{attribute 'GeneratedUsingTerminal: IODEVICETYPE_ETHERCATPROT'}
{attribute addProperty BoxType "IODEVICETYPE_ETHERCATPROT"}
{attribute addProperty Id "Beckhoff_EL1xxxBeckhoff_EL1xxx_3E37AACA6236Beckhoff_EL2xxxBeckhoff_EL2xxx_F4C539CA2992Beckhoff_EL3xxxBeckhoff_EL3xxx_05984D3D1813Beckhoff_EL3xxx_0030Beckhoff_EL3xxx_0030_C37B7D48265Beckhoff_EL4xxxBeckhoff_EL4xxx_44DCAF8D2405Beckhoff_EL5xxxBeckhoff_EL5xxx_A510F2723086Beckhoff_EL6xxxBeckhoff_EL6xxx_5832F4A84115Beckhoff_EL7xxxBeckhoff_EL7xxx_96878FD52666Beckhoff_EL9xxxBeckhoff_EL9xxx_6E572B5F1254Beckhoff_EL15xxBeckhoff_EL15xx_7FFDF3B3529Beckhoff_EL19xxBeckhoff_EL19xx_C9550BF750Beckhoff_EL25xxBeckhoff_EL25xx_A1E3F9182720Beckhoff_EL29xxBeckhoff_EL29xx_FCC67B4476Beckhoff_EL30xxBeckhoff_EL30xx_59D865295129Beckhoff_EL31xxBeckhoff_EL31xx_098DC56E3694Beckhoff_EL32xxBeckhoff_EL32xx_A91E9D412581Beckhoff_EL33xxBeckhoff_EL33xx_149C8FF52459Beckhoff_EL34xxBeckhoff_EL34xx_5C8507D711825Beckhoff_EL37xxBeckhoff_EL37xx_82AB11DA2253Beckhoff_EL47xxBeckhoff_EL47xx_F9F61196294Beckhoff_EL66xxBeckhoff_EL66xx_32F43B791034Beckhoff_EL67xxBeckhoff_EL67xx_9D033AAA966Beckhoff_EL68xxBeckhoff_EL68xx_6F2062753597Beckhoff_EL69xxBeckhoff_EL69xx_55DE5C9C198Beckhoff_EL72xxBeckhoff_EL72xx_566ED46D3383Beckhoff_EL73xxBeckhoff_EL73xx_3D4E24E01278Beckhoff_EL99xxBeckhoff_EL99xx_FA66A12D10SyncUnitsSyncUnits_9F8710E11242InputsInputs_25A0042B160OutputsOutputs_2397A10E106InfoDataInfoData_E68C61CD28"}
{attribute addProperty CRC "3501869254"}
{attribute addProperty Size "68444"}
TYPE EtherCAT_Master_ELxxxx_D0BA48C6 EXTENDS EtcMasterBase_62654B43 :
STRUCT
	{attribute addProperty Name "Beckhoff EL1xxx"}
	{attribute addProperty PreviousPort "EtherCAT_Master_ELxxxx : Master"}
	Beckhoff_EL1xxx : Beckhoff_EL1xxx_3E37AACA;
	{attribute addProperty Name "Beckhoff EL2xxx"}
	{attribute addProperty PreviousPort "Beckhoff EL1xxx : C"}
	Beckhoff_EL2xxx : Beckhoff_EL2xxx_F4C539CA;
	{attribute addProperty Name "Beckhoff EL3xxx"}
	{attribute addProperty PreviousPort "Beckhoff EL2xxx : C"}
	Beckhoff_EL3xxx : Beckhoff_EL3xxx_05984D3D;
	{attribute addProperty Name "Beckhoff EL3xxx-0030"}
	{attribute addProperty PreviousPort "Beckhoff EL3xxx : C"}
	Beckhoff_EL3xxx_0030 : Beckhoff_EL3xxx_0030_C37B7D48;
	{attribute addProperty Name "Beckhoff EL4xxx"}
	{attribute addProperty PreviousPort "Beckhoff EL3xxx-0030 : C"}
	Beckhoff_EL4xxx : Beckhoff_EL4xxx_44DCAF8D;
	{attribute addProperty Name "Beckhoff EL5xxx"}
	{attribute addProperty PreviousPort "Beckhoff EL4xxx : C"}
	Beckhoff_EL5xxx : Beckhoff_EL5xxx_A510F272;
	{attribute addProperty Name "Beckhoff EL6xxx"}
	{attribute addProperty PreviousPort "Beckhoff EL5xxx : C"}
	Beckhoff_EL6xxx : Beckhoff_EL6xxx_5832F4A8;
	{attribute addProperty Name "Beckhoff EL7xxx"}
	{attribute addProperty PreviousPort "Beckhoff EL6xxx : C"}
	Beckhoff_EL7xxx : Beckhoff_EL7xxx_96878FD5;
	{attribute addProperty Name "Beckhoff EL9xxx"}
	{attribute addProperty PreviousPort "Beckhoff EL7xxx : C"}
	Beckhoff_EL9xxx : Beckhoff_EL9xxx_6E572B5F;
	{attribute addProperty Name "Beckhoff EL15xx"}
	{attribute addProperty PreviousPort "Beckhoff EL9xxx : C"}
	Beckhoff_EL15xx : Beckhoff_EL15xx_7FFDF3B3;
	{attribute addProperty Name "Beckhoff EL19xx"}
	{attribute addProperty PreviousPort "Beckhoff EL15xx : C"}
	Beckhoff_EL19xx : Beckhoff_EL19xx_C9550BF7;
	{attribute addProperty Name "Beckhoff EL25xx"}
	{attribute addProperty PreviousPort "Beckhoff EL19xx : C"}
	Beckhoff_EL25xx : Beckhoff_EL25xx_A1E3F918;
	{attribute addProperty Name "Beckhoff EL29xx"}
	{attribute addProperty PreviousPort "Beckhoff EL25xx : C"}
	Beckhoff_EL29xx : Beckhoff_EL29xx_FCC67B44;
	{attribute addProperty Name "Beckhoff EL30xx"}
	{attribute addProperty PreviousPort "Beckhoff EL29xx : C"}
	Beckhoff_EL30xx : Beckhoff_EL30xx_59D86529;
	{attribute addProperty Name "Beckhoff EL31xx"}
	{attribute addProperty PreviousPort "Beckhoff EL30xx : C"}
	Beckhoff_EL31xx : Beckhoff_EL31xx_098DC56E;
	{attribute addProperty Name "Beckhoff EL32xx"}
	{attribute addProperty PreviousPort "Beckhoff EL31xx : C"}
	Beckhoff_EL32xx : Beckhoff_EL32xx_A91E9D41;
	{attribute addProperty Name "Beckhoff EL33xx"}
	{attribute addProperty PreviousPort "Beckhoff EL32xx : C"}
	Beckhoff_EL33xx : Beckhoff_EL33xx_149C8FF5;
	{attribute addProperty Name "Beckhoff EL34xx"}
	{attribute addProperty PreviousPort "Beckhoff EL33xx : C"}
	Beckhoff_EL34xx : Beckhoff_EL34xx_5C8507D7;
	{attribute addProperty Name "Beckhoff EL37xx"}
	{attribute addProperty PreviousPort "Beckhoff EL34xx : C"}
	Beckhoff_EL37xx : Beckhoff_EL37xx_82AB11DA;
	{attribute addProperty Name "Beckhoff EL47xx"}
	{attribute addProperty PreviousPort "Beckhoff EL37xx : C"}
	Beckhoff_EL47xx : Beckhoff_EL47xx_F9F61196;
	{attribute addProperty Name "Beckhoff EL66xx"}
	{attribute addProperty PreviousPort "Beckhoff EL47xx : C"}
	Beckhoff_EL66xx : Beckhoff_EL66xx_32F43B79;
	{attribute addProperty Name "Beckhoff EL67xx"}
	{attribute addProperty PreviousPort "Beckhoff EL66xx : C"}
	Beckhoff_EL67xx : Beckhoff_EL67xx_9D033AAA;
	{attribute addProperty Name "Beckhoff EL68xx"}
	{attribute addProperty PreviousPort "Beckhoff EL67xx : C"}
	Beckhoff_EL68xx : Beckhoff_EL68xx_6F206275;
	{attribute addProperty Name "Beckhoff EL69xx"}
	{attribute addProperty PreviousPort "Beckhoff EL68xx : C"}
	Beckhoff_EL69xx : Beckhoff_EL69xx_55DE5C9C;
	{attribute addProperty Name "Beckhoff EL72xx"}
	{attribute addProperty PreviousPort "Beckhoff EL69xx : C"}
	Beckhoff_EL72xx : Beckhoff_EL72xx_566ED46D;
	{attribute addProperty Name "Beckhoff EL73xx"}
	{attribute addProperty PreviousPort "Beckhoff EL72xx : C"}
	Beckhoff_EL73xx : Beckhoff_EL73xx_3D4E24E0;
	{attribute addProperty Name "Beckhoff EL99xx"}
	{attribute addProperty PreviousPort "Beckhoff EL73xx : C"}
	Beckhoff_EL99xx : Beckhoff_EL99xx_FA66A12D;
	{attribute addProperty Name "SyncUnits"}
	SyncUnits : SyncUnits_9F8710E1;
	{attribute addProperty Name "Inputs"}
	Inputs : Inputs_25A0042B;
	{attribute addProperty Name "Outputs"}
	Outputs : Outputs_2397A10E;
	{attribute addProperty Name "InfoData"}
	InfoData : InfoData_E68C61CD;
END_STRUCT
END_TYPE

(* stored: Version 1.2.0.0, ProductVersion 3.1.4024.9
   DUT EtherCAT_Master_ELxxxx_D0BA48C6: Id {babc382e-0a00-46d6-b0c5-b46fe6b45e49} *)
